TYPE ST_VRC EXTENDS ST_ValveBase:
STRUCT
(* Readbacks *)
	//In case VRC is normally open
	{attribute 'pytmc' := '
    pv: CLS_OK;
	io: i;
    '}
	xCLS_OK : BOOL := TRUE;

END_STRUCT
END_TYPE

(* stored: Version 1.1.0.1, ProductVersion 3.1.4022.18
   DUT ST_VRC: Id {ee6efa67-7be0-4e42-b045-50546d4578bb} *)
